// TIA Portal V17 export
// export: Created 2022-03-12T16:05:31.627286Z, ExportSetting WithDefaults, DisplayName Totally Integrated Automation Portal, DisplayVersion V17, DisplayName TIA Portal Openness, DisplayVersion V17, DisplayName TIA Portal Version Control Interface, DisplayVersion V17, DisplayName STEP 7 Professional, DisplayVersion V17, DisplayName STEP 7 Safety, DisplayVersion V17, DisplayName WinCC Advanced / Unified PC, DisplayVersion V17
DATA_BLOCK "ParetoData"   // DB31617
TITLE = CPG_ParetoData
{ S7_Optimized_Access := 'TRUE' }
AUTHOR : tech.team.motioncontrol@siemens.com
FAMILY : CPG
VERSION : 1.1
// Support: tech.team.motioncontrol@siemens.com
// stored: AutoNumber true, DBAccessibleFromOPCUA true, DBAccessibleFromWebserver true, IsOnlyStoredInLoadMemory false, IsRetainMemResEnabled false, IsWriteProtectedInAS false, MemoryReserve 0
   VAR RETAIN
      alarmOccurrence { S7_SetPoint := 'True'} : Array[0.."CPG_PARTEO_NO_OF_ERRORS_UPPER_LIM"] of "CPG_typePareto";   // Alarm Array
      totalStops : Int;   // Total stops on the machine
      totalTimeSinceReset : Real;   // Total time since reset
      totalUptime : Real;   // Total uptime of the machine
      totalDowntime : Real;   // Total downtime of the machine
      percentUptime : Real;
      MTTR : Real;
      MTBF : Real;
      Sort : Int;
      Reset : Bool;
   END_VAR
BEGIN
END_DATA_BLOCK
